TEXTLIST ModeRowText
  10000 = 'Power On' | 汉语: '汉语'
  10001 = 'Power On' | 汉语: '汉语'
  10002 = '10002' | 汉语: '汉语'
  10003 = 'Power Off' | 汉语: '汉语'
  10004 = 'Power Off' | 汉语: '汉语'
  10005 = '10005'
  10006 = 'Power'
  10007 = '10007'
  10008 = '10008'
  10009 = '10009'
  10010 = '10010'
  10011 = '10011'
  10012 = '10012'
  10013 = '10013'
  10014 = '10014'
  10015 = '10015'
  10016 = '10016'
  10017 = '10017'
  10018 = '10018'
  10019 = '10019'
  10020 = 'Automatic'
  10021 = 'Automatic'
  10022 = '10022'
  10023 = 'Manual'
  10024 = 'Manual'
  10025 = '10025'
  10026 = 'Mode'
  10027 = '10027'
  10028 = '10028'
  10029 = '10029'
  10030 = '10030'
  10031 = '10031'
  10032 = '10032'
  10033 = '10033'
  10034 = '10034'
  10035 = '10035'
  10036 = '10036'
  10037 = '10037'
  10038 = '10038'
  10039 = '10039'
  10040 = 'Continuous Cycle'
  10041 = 'Continuous Cycle'
  10042 = '10042'
  10043 = 'Single Cycle'
  10044 = 'Single Cycle'
  10045 = '10045'
  10046 = 'Cycle'
  10047 = '10047'
  10048 = '10048'
  10049 = '10049'
  10050 = '10050'
  10051 = '10051'
  10052 = '10052'
  10053 = '10053'
  10054 = '10054'
  10055 = '10055'
  10056 = '10056'
  10057 = '10057'
  10058 = '10058'
  10059 = '10059'
  10060 = 'Auto Cycle Start'
  10061 = 'Auto Cycling'
  10062 = '10062'
  10063 = 'Stop Cycle'
  10064 = 'Auto Cycle Stopped'
  10065 = '10065'
  10066 = 'Cycle Start'
  10067 = '10067'
  10068 = '10068'
  10069 = '10069'
  10070 = '10070'
  10071 = '10071'
  10072 = '10072'
  10073 = '10073'
  10074 = '10074'
  10075 = '10075'
  10076 = '10076'
  10077 = '10077'
  10078 = '10078'
  10079 = '10079'
  10080 = '10080'
  10081 = '10081'
  10082 = '10082'
  10083 = 'Return Home'
  10084 = 'Home'
  10085 = '10085'
  10086 = 'Home'
  10087 = '10087'
  10088 = '10088'
  10089 = '10089'
  10090 = '10090'
  10091 = '10091'
  10092 = '10092'
  10093 = '10093'
  10094 = '10094'
  10095 = '10095'
  10096 = '10096'
  10097 = '10097'
  10098 = '10098'
  10099 = '10099'
  10100 = 'To Wash Posn'
  10101 = 'At Wash Posn'
  10102 = '10102'
  10103 = 'To Place Pounce'
  10104 = 'At Place Pounce'
  10105 = '10105'
  10106 = 'Robot'
  10107 = '10107'
  10108 = '10108'
  10109 = '10109'
  10110 = '10110'
  10111 = '10111'
  10112 = '10112'
  10113 = '10113'
  10114 = '10114'
  10115 = '10115'
  10116 = '10116'
  10117 = '10117'
  10118 = '10118'
  10119 = '10119'
  10120 = 'Start Washer'
  10121 = 'Washer On'
  10122 = '10122'
  10123 = 'Stop Washer'
  10124 = 'Washer Off'
  10125 = '10125'
  10126 = 'Washer Jets'
  10127 = '10127'
  10128 = '10128'
  10129 = '10129'
  10130 = '10130'
  10131 = '10131'
  10132 = '10132'
  10133 = '10133'
  10134 = '10134'
  10135 = '10135'
  10136 = '10136'
  10137 = '10137'
  10138 = '10138'
  10139 = '10139'
  10140 = '10140'
  10141 = '10141'
  10142 = '10142'
  10143 = 'Lock'
  10144 = 'Locked'
  10145 = '10145'
  10146 = 'Access Door'
  10147 = '10147'
  10148 = '10148'
  10149 = '10149'
  10150 = '10150'
  10151 = '10151'
  10152 = '10152'
  10153 = '10153'
  10154 = '10154'
  10155 = '10155'
  10156 = '10156'
  10157 = '10157'
  10158 = '10158'
  10159 = '10159'
  10160 = 'Request Access Gate 1'
  10161 = 'Request Access Gate 1'
  10162 = '10162'
  10163 = 'Request Access Gate 2'
  10164 = 'Request Access Gate 2'
  10165 = '10165'
  10166 = 'Access Door'
  10167 = '10167'
  10168 = '10168'
  10169 = '10169'
  10170 = '10170'
  10171 = '10171'
  10172 = '10172'
  10173 = '10173'
  10174 = '10174'
  10175 = '10175'
  10176 = '10176'
  10177 = '10177'
  10178 = '10178'
  10179 = '10179'
  10180 = '10180'
  10181 = '10181'
  10182 = '10182'
  10183 = '10183'
  10184 = '10184'
  10185 = '10185'
  10186 = '10186'
  10187 = '10187'
  10188 = '10188'
  10189 = '10189'
  10190 = '10190'
  10191 = '10191'
  10192 = '10192'
  10193 = '10193'
  10194 = '10194'
  10195 = '10195'
  10196 = '10196'
  10197 = '10197'
  10198 = '10198'
  10199 = '10199'
   = ''
END_TEXTLIST

(* stored: Version 1.1.0.1, ProductVersion 3.1.4024.12
   TextList ModeRowText: Id {d23a3f5b-47f0-458b-b35b-3475d69b8114} *)
